// TIA Portal V18 export
FUNCTION "AHUSupplyFanCtrl" : Void   // FC60302, LAD
{ S7_Optimized_Access := 'TRUE' }
VERSION : 0.1
// Cfg
// 0 - No Fan (No AHU)
// 1 - Adaptation/Proxi
// 2 - 1Speed
// 3 - 2Speed
// 4 - 0-100%
// stored: AutoNumber false, IsIECCheckEnabled false, SetENOAutomatically false, UDAEnableTagReadback false
   VAR_INPUT
      iUnitID : Int;
      cFanUnitCfg : Byte;
      xFanBlocking : Bool;
      rDemandFreshAir : Real;
      rDemandHeating : Real;
      rDemandCooling : Real;
      rDemandFrostProtection : Real;
      xDieselOperation : Bool;
      rFanAOCoefDieselOperation : Real;
      rFanAOCoefGridOperation : Real;
   END_VAR
   VAR_IN_OUT
      rFanSpeedAORequest : Real;
      xFanSpeedAOEnable : Bool;
      xSpeed2DORequest : Bool;
      xSpeed1DORequest : Bool;
   END_VAR
   VAR_TEMP
      rSumDemand : Real;
      rSumDemandInt1 : Real;
      rSumDemandInt2 : Real;
      rRawFanAO : Real;
      xRawFanSt1Request : Bool;
      xRawFanSt2Request : Bool;
      xRawFanAOEnable : Bool;
   END_VAR
BEGIN

REGION Network 1 (SCL)
   CASE #cFanUnitCfg OF
       0:  // No Unit
           ;
       1:  // Proxy
           ;
       2:   // Single speed
           ; 
       3:   // Two speed fan motor
           ;
       4:  // 0-100% Modulative
           #xSpeed1DORequest := 0;
           #xSpeed2DORequest := 0;

           IF #xFanBlocking THEN
               #rRawFanAO := 0;
               #xFanSpeedAOEnable := 0;
           ELSE
               #rSumDemandInt1 := MAX(IN1 := #rDemandFreshAir, IN2 := #rDemandHeating);
               #rSumDemandInt2 := MAX(IN1 := #rDemandFrostProtection, IN2 := #rDemandCooling);
               #rSumDemand := MAX(IN1 := #rSumDemandInt1, IN2 := #rSumDemandInt2);

               IF #rSumDemand > 5 THEN
                   #rFanSpeedAORequest := 1;
                   #rRawFanAO := #rSumDemand;
               ELSIF #rSumDemand < 1 THEN
                   #rFanSpeedAORequest := 0;
                   #xFanSpeedAOEnable := 0;
               END_IF;
           END_IF;
           ;
       ELSE  // Statement section ELSE
           ;
   END_CASE;
END_REGION

REGION Network 2 (SCL)
   IF #xDieselOperation THEN
       #xSpeed2DORequest := 0;
       #xSpeed1DORequest := #xRawFanSt1Request OR #xRawFanSt2Request;
       #rFanSpeedAORequest := #rRawFanAO * #rFanAOCoefDieselOperation;
       #xFanSpeedAOEnable := #xRawFanAOEnable;
   END_IF;
END_REGION
END_FUNCTION
